// TIA Portal project "motor_uygulamasi_2" (V18)

(* hardware
DEVICE "S7-1200 station_1"  S7-1200 Station
   slot 0: "Rack_0"  S7-1200 Rack  Rack  V1.0
   slot 1: "PLC_1"  CPU 1214C AC/DC/Rly  6ES7 214-1BG40-0XB0  V4.6
*)

// ===== PLC "PLC_1"  CPU 1214C AC/DC/Rly =====

VAR_GLOBAL   // PLC tag table "Default tag table"
   "STOP" AT %I0.0 : Bool;
   "LS1" AT %I0.1 : Bool;
   "MOTOR2" AT %Q0.2 : Bool;
   "MOTOR1" AT %Q0.1 : Bool;
END_VAR

ORGANIZATION_BLOCK "Main"   // OB1, LAD, ProgramCycle
TITLE = "Main Program Sweep (Cycle)"
{ S7_Optimized_Access := 'TRUE' }
VERSION : 0.1
// UYGULAMA-2: Bir sistem, 1 adet sinir anahtar ve bir adet stop butonu ile kumanda edilecektir. Mekanik bir sistem gelip sinIr
// anahtarina carptiginda 1. motor surekli, 2. motor ise hareketli sistem sinir anahtarina bask wyguladigi strece devrede kalacaktir.
// Mekanik sistem sinir anahtarindan kurtuldugu anda 2. motor duracak, 1. motor alismaya devam edecektir. Stop butonuna
// basildiginda tüm sistem duracaktir.
   VAR_INPUT
      Initial_Call : Bool;   // Initial call of this OB
      Remanence : Bool;   // =True, if remanent data are available
   END_VAR
BEGIN

REGION Network 1
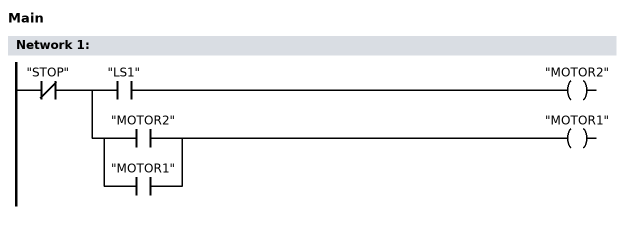
   RUNG wire#powerrail
      I_Contact( "STOP" )
      wire#w1
      Contact( "LS1" )
      Coil( "MOTOR2" )
   END_RUNG
   RUNG wire#w1
      Contact( "MOTOR2" )
      wire#w2
      Coil( "MOTOR1" )
   END_RUNG
   RUNG wire#w1
      Contact( "MOTOR1" )
   END_RUNG wire#w2
   // the same network as SCL:
   "MOTOR2" := NOT "STOP" AND "LS1";
   "MOTOR1" := NOT "STOP" AND ("MOTOR2" OR "MOTOR1");
END_REGION
END_ORGANIZATION_BLOCK